(* IEC 61131-3 sources: CodesysTest/export/Function Blocks/FB_BaseComponent.pou, 4 files *)

(* ---- FB_BaseComponent.pou.st ---- *)
(*#-#-#-#-#-#-#-#-#-#---Declaration---#-#-#-#-#-#-#-#-#-#-#-#-#*)

FUNCTION_BLOCK FB_BaseComponent EXTENDS FB_BaseObject IMPLEMENTS IComponent, IMachineOption, IExecuteAutomatically
VAR_INPUT
END_VAR
VAR_OUTPUT

END_VAR
VAR
    _ready : BOOL;                    // Ready to be controlled
	_reset : BOOL;
	_optionActive : BOOL;
	_optionEnabled : BOOL;
	_optionInstalled : BOOL;
	enableONS : R_TRIG;
	resetONS : R_TRIG;
END_VAR
(*#-#-#-#-#-#-#-#-#-#---Implementation---#-#-#-#-#-#-#-#-#-#-#-#-#*)

//	Function Block: BaseComponentFB
//	Description:  Extend this FB for each component as it contains the basic variables and logic that all components must share
//	In all extended FBs that have an Execute() method you must run the parent logic with SUPER^()
//	Created by: Ben Hess
//	Created Date: Friday, June 1, 2018

_optionActive := _optionEnabled AND _optionInstalled;

(* ---- Execute.m.st ---- *)
(*#-#-#-#-#-#-#-#-#-#---Declaration---#-#-#-#-#-#-#-#-#-#-#-#-#*)

METHOD Execute
VAR_INPUT
END_VAR
(*#-#-#-#-#-#-#-#-#-#---Implementation---#-#-#-#-#-#-#-#-#-#-#-#-#*)

_optionActive := _optionEnabled AND _optionInstalled;

(* ---- MakeReady.m.st ---- *)
(*#-#-#-#-#-#-#-#-#-#---Declaration---#-#-#-#-#-#-#-#-#-#-#-#-#*)

METHOD MakeReady : BOOL
VAR_INPUT
END_VAR
(*#-#-#-#-#-#-#-#-#-#---Implementation---#-#-#-#-#-#-#-#-#-#-#-#-#*)

_makeReady := TRUE;

(* ---- SterilizeVariables.m.st ---- *)
(*#-#-#-#-#-#-#-#-#-#---Declaration---#-#-#-#-#-#-#-#-#-#-#-#-#*)

METHOD SterilizeVariables : BOOL
VAR_INPUT
END_VAR
(*#-#-#-#-#-#-#-#-#-#---Implementation---#-#-#-#-#-#-#-#-#-#-#-#-#*)

//This Method will be used to reset all variables to what they should be in the idle state.  should be called whenever we want to make sure all variables are in a known condition.
